// TIA Portal V17 export
// export: Created 2023-02-13T11:16:47.778915Z, ExportSetting WithDefaults, DisplayName Totally Integrated Automation Portal, DisplayVersion V17, DisplayName TIA Portal Openness, DisplayVersion V17, DisplayName TIA Portal Teamcenter Gateway, DisplayVersion V17, DisplayName TIA Portal Version Control Interface, DisplayVersion V17, DisplayName SINAMICS Startdrive Advanced, DisplayVersion V17, DisplayName SINAMICS Startdrive G130, G150, S120, S150, SINAMICS MV, S210, DisplayVersion V17, DisplayName SINAMICS Startdrive G110M, G120, G120C, G120D, G120P, G115D, DisplayVersion V17, DisplayName STEP 7 Professional, DisplayVersion V17, DisplayName STEP 7 Safety, DisplayVersion V17, DisplayName WinCC Professional, DisplayVersion V17
FUNCTION_BLOCK "Raw_Pulse"   // FB20, LAD
{ S7_Optimized_Access := 'TRUE' }
VERSION : 0.1
// stored: AutoNumber true, IsIECCheckEnabled false, IsRetainMemResEnabled false, MemoryReserve 100, SetENOAutomatically false, UDAEnableTagReadback false
   VAR_INPUT
      CountReset : Bool;
      CountMode : Bool;
      DoseRun : Bool;
      CmdStep : Int;
      FT_Pulse : Bool;   // Pulse Flow Meter
      FT_Tot : Real;
      Dose_SP : Real;
      Speed_AV : Real;
      Speed_SP : Real;
   END_VAR
   VAR_OUTPUT
      Q_FT_Star : Real;
      Q_FT_Stop : Real;
      Q_SPQty : Real;
      Q_FineQty : Real;
      Q_StopQty : Real;
      Q_P_Speed : Real;
      Q_P_FineSpeed : Real;
      Q_P_CoasSpeed : Real;
   END_VAR
   VAR_IN_OUT
      Q_FT_Tot : Real;
   END_VAR
   VAR RETAIN
      Para : Struct
         "SP_Qty_Stop%" : Real := 3.0;
         "SP_Qty_Fine%" : Real := 20.0;
         SP_Qty_Stop : Real;
         SP_Qty_Fine : Real;
         SP_Pump_Co : Real := 80.0;
         SP_Pump_Fi : Real := 20.0;
         "Pulse/Liter" : Real := 1.0;
      END_STRUCT;
   END_VAR
   VAR
      alwaysON { S7_SetPoint := 'True'} : Bool;
      DosePE : Bool;
      "BIT.FT_Pulse" : Bool;
   END_VAR
   VAR_TEMP   // added for the SCL form of the ladder/FBD networks
      _w1 : Bool;
      _w2 : Bool;
      _w3 : Bool;
      _w4 : Bool;
   END_VAR
BEGIN

REGION Network 1: alwaysON
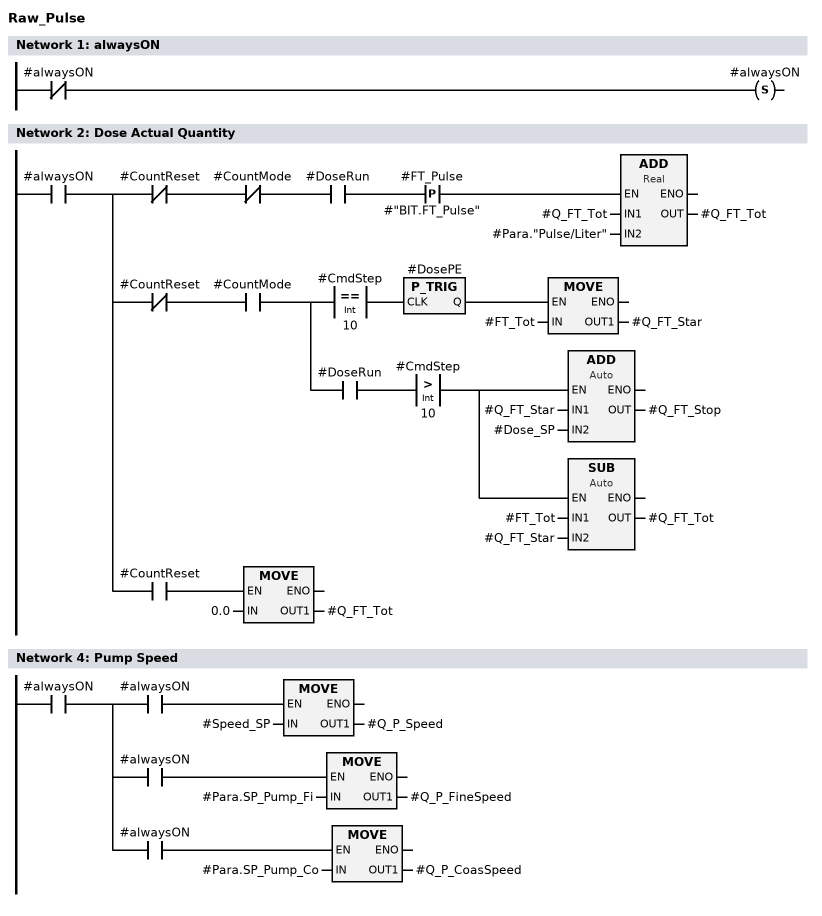
   RUNG wire#powerrail
      I_Contact( #alwaysON )
      S_Coil( #alwaysON )
   END_RUNG
   // the same network as SCL:
   IF NOT #alwaysON THEN #alwaysON := TRUE; END_IF;
END_REGION

REGION Network 2: Dose Actual Quantity
   RUNG wire#powerrail
      Contact( #alwaysON )
      wire#w1
      I_Contact( #CountReset )
      I_Contact( #CountMode )
      Contact( #DoseRun )
      P_Contact(operand := #FT_Pulse, bit := #"BIT.FT_Pulse")
      { S7_Templates := "SrcType := Real" } Add(in1 := #Q_FT_Tot, in2 := #Para."Pulse/Liter", out => #Q_FT_Tot)
   END_RUNG
   RUNG wire#w1
      I_Contact( #CountReset )
      Contact( #CountMode )
      wire#w2
      { S7_Templates := "SrcType := Int" } EQ_Contact(in1 := #CmdStep, in2 := 10)
      P_Trig( #DosePE )
      Move(in := #FT_Tot, out1 => #Q_FT_Star)
   END_RUNG
   RUNG wire#w2
      Contact( #DoseRun )
      { S7_Templates := "SrcType := Int" } GT_Contact(in1 := #CmdStep, in2 := 10)
      wire#w3
      Add(in1 := #Q_FT_Star, in2 := #Dose_SP, out => #Q_FT_Stop)
   END_RUNG
   RUNG wire#w3
      Sub(in1 := #FT_Tot, in2 := #Q_FT_Star, out => #Q_FT_Tot)
   END_RUNG
   RUNG wire#w1
      Contact( #CountReset )
      Move(in := 0.0, out1 => #Q_FT_Tot)
   END_RUNG
   // the same network as SCL:
   #_w1 := #alwaysON AND NOT #CountReset AND NOT #CountMode AND #DoseRun AND #FT_Pulse AND NOT #"BIT.FT_Pulse";   // rising edge of #FT_Pulse
   #"BIT.FT_Pulse" := #FT_Pulse;
   IF #_w1 THEN #Q_FT_Tot := #Q_FT_Tot + #Para."Pulse/Liter"; END_IF;
   #_w2 := #alwaysON AND NOT #CountReset AND #CountMode;
   #_w3 := #_w2 AND (#CmdStep = 10);
   #_w4 := #_w3 AND NOT #DosePE;   // rising edge
   #DosePE := #_w3;
   IF #_w4 THEN #Q_FT_Star := #FT_Tot; END_IF;
   IF #_w2 AND #DoseRun AND (#CmdStep > 10) THEN
       #Q_FT_Stop := #Q_FT_Star + #Dose_SP;
       #Q_FT_Tot := #FT_Tot - #Q_FT_Star;
   END_IF;
   IF #alwaysON AND #CountReset THEN #Q_FT_Tot := 0.0; END_IF;
END_REGION

NETWORK
TITLE = Quantity Calculation
// SP Quantity
      L     #Dose_SP;
      T     #Q_SPQty;
// Fine Quantity Calculation
      L     #Dose_SP;
      L     #Para."SP_Qty_Fine%";
      *R;
      L     100.0;
      /R;
      T     #Para.SP_Qty_Fine;

      L     #Dose_SP;
      L     #Para.SP_Qty_Fine;
      -R;
      T     #Q_FineQty;

// Stop Quantity Calculation
      L     #Dose_SP;
      L     #Para."SP_Qty_Stop%";
      *R;
      L     100.0;
      /R;
      T     #Para.SP_Qty_Stop;

      L     #Dose_SP;
      L     #Para.SP_Qty_Stop;
      -R;
      T     #Q_StopQty;


REGION Network 4: Pump Speed
   RUNG wire#powerrail
      Contact( #alwaysON )
      wire#w1
      Contact( #alwaysON )
      Move(in := #Speed_SP, out1 => #Q_P_Speed)
   END_RUNG
   RUNG wire#w1
      Contact( #alwaysON )
      Move(in := #Para.SP_Pump_Fi, out1 => #Q_P_FineSpeed)
   END_RUNG
   RUNG wire#w1
      Contact( #alwaysON )
      Move(in := #Para.SP_Pump_Co, out1 => #Q_P_CoasSpeed)
   END_RUNG
   // the same network as SCL:
   IF #alwaysON AND #alwaysON THEN
       #Q_P_Speed := #Speed_SP;
       #Q_P_FineSpeed := #Para.SP_Pump_Fi;
       #Q_P_CoasSpeed := #Para.SP_Pump_Co;
   END_IF;
END_REGION
END_FUNCTION_BLOCK
